// TIA Portal V17 export
// export: Created 2022-02-03T14:45:13.7246224Z, ExportSetting WithDefaults, DisplayName Totally Integrated Automation Portal, DisplayVersion V17, DisplayName TIA Portal Openness, DisplayVersion V17, DisplayName TIA Portal Version Control Interface, DisplayVersion V17, DisplayName SINAMICS Startdrive Advanced, DisplayVersion V17, DisplayName SINAMICS Startdrive G130, G150, S120, S150, SINAMICS MV, S210, DisplayVersion V17, DisplayName SINAMICS Startdrive G110M, G120, G120C, G120D, G120P, G115D, DisplayVersion V17, DisplayName STEP 7 Professional, DisplayVersion V17, DisplayName STEP 7 Safety, DisplayVersion V17, DisplayName WinCC Advanced, DisplayVersion V17
DATA_BLOCK "NewWeightToStore_DB"   // DB11
VERSION : 0.1
// stored: Access Unpublished, AutoNumber true, DBAccessibleFromOPCUA true, DBAccessibleFromWebserver true, InstanceOfName NewWeightToStore, InstanceOfType FB
"NewWeightToStore"
   // VAR_INPUT
   //    occupiedBay : Array["FIRSTBAY".."LASTBAY"] of Bool;
   //    weightBay : Array["FIRSTBAY".."LASTBAY"] of UInt;
   //    initStore : Bool;
   //    storeNo : UInt;
   //    initAllStores : Bool;
   // END_VAR
   // VAR_OUTPUT
   //    storeFull : Bool;
   // END_VAR
   // VAR_IN_OUT
   //    store : Array[0..9] of "typeStore";
   //    storeStatistics : "typeStoreStatistics";
   // END_VAR
   // VAR
   //    statOldOccupiedBay : Array["FIRSTBAY".."LASTBAY"] of Bool;
   //    statOldInitStore : Bool;
   //    statStoreNo : UInt;
   // END_VAR
BEGIN
END_DATA_BLOCK
